FUNCTION_BLOCK INT_TO_BIT (* Basic Function Block Type *)
  (* Standard: 61499-2 *)
  (* Version 0.0, 27/11/2020, Schulung, Schneider Electric, Template *)
  PACKAGE Main;
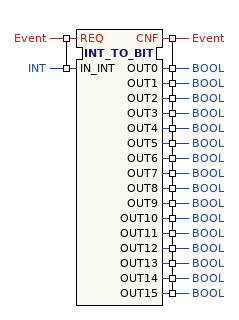
  EVENT_INPUT
    REQ WITH IN_INT; (* Normal Execution Request *)
  END_EVENT
  EVENT_OUTPUT
    CNF WITH OUT0, OUT1, OUT2, OUT3, OUT4, OUT5, OUT6, OUT7, OUT8, OUT9, OUT10, OUT11, OUT12, OUT13, OUT14, OUT15; (* Execution Confirmation *)
  END_EVENT
  VAR_INPUT
    IN_INT : INT; (* Input event qualifier *)
  END_VAR
  VAR_OUTPUT
    OUT0 : BOOL; (* Output event qualifier *)
    OUT1 : BOOL;
    OUT2 : BOOL;
    OUT3 : BOOL;
    OUT4 : BOOL;
    OUT5 : BOOL;
    OUT6 : BOOL;
    OUT7 : BOOL;
    OUT8 : BOOL;
    OUT9 : BOOL;
    OUT10 : BOOL;
    OUT11 : BOOL;
    OUT12 : BOOL;
    OUT13 : BOOL;
    OUT14 : BOOL;
    OUT15 : BOOL;
  END_VAR
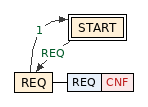
  EC_STATES
    START; (* Initial State *)
    REQ : REQ -> CNF; (* Normal execution *)
  END_STATES
  EC_TRANSITIONS
    START TO REQ := REQ;
    REQ TO START := 1;
  END_TRANSITIONS
  ALGORITHM REQ IN ST: (* Normally executed algorithm *)
OUT0 := EQ(AND(IN_INT,16#0001),16#0001);
OUT1 := EQ(AND(IN_INT,16#0002),16#0002);
OUT2 := EQ(AND(IN_INT,16#0004),16#0004);
OUT3 := EQ(AND(IN_INT,16#0008),16#0008);
OUT4 := EQ(AND(IN_INT,16#0010),16#0010);
OUT5 := EQ(AND(IN_INT,16#0020),16#0020);
OUT6 := EQ(AND(IN_INT,16#0040),16#0040);
OUT7 := EQ(AND(IN_INT,16#0080),16#0080);
OUT8 := EQ(AND(IN_INT,16#0100),16#0100);
OUT9 := EQ(AND(IN_INT,16#0200),16#0200);
OUT10 := EQ(AND(IN_INT,16#0400),16#0400);
OUT11 := EQ(AND(IN_INT,16#0800),16#0800);
OUT12 := EQ(AND(IN_INT,16#1000),16#1000);
OUT13 := EQ(AND(IN_INT,16#2000),16#2000);
OUT14 := EQ(AND(IN_INT,16#4000),16#4000);
OUT15 := EQ(AND(INT_TO_WORD(IN_INT),16#8000),16#8000);
  END_ALGORITHM
END_FUNCTION_BLOCK
